PROGRAM MAIN
VAR
	bPizzaInOven : BOOL;
	fbMyTimer	 : TON;
	fbMyTrigger_RTRIG : R_TRIG;
	bBuzzer 	 : BOOL;
	iTotalPizzasCooked	: UDINT;
END_VAR

fbMyTimer(IN:=bPizzaInOven,PT := T#3S);

bBuzzer := fbMyTimer.Q;

fbMyTrigger_RTRIG(clk:=fbMyTimer.Q);

IF fbMyTrigger_RTRIG.Q THEN
	iTotalPizzasCooked := iTotalPizzasCooked + 1;
END_IF

END_PROGRAM

(* stored: Version 1.1.0.1, ProductVersion 3.1.4019.2
   POU MAIN: Id {ac7b629d-ed59-42db-ae7f-63afec425186}, SpecialFunc None *)
